{attribute 'linkalways'} 
{attribute 'no_explicit_call' := 'This FB is a CLASS and must be accessed using methods or properties'}
{attribute 'enable_dynamic_creation'}
FUNCTION_BLOCK Node_F_VN_ScharrFilter EXTENDS VisionNode
VAR
	ipSrcImage : _ITcVnImage;
    ipDestImage : _ITcVnImage;
    eDestDepth : _ETcVnElementType(ETcVnElementType.TCVN_ET_SAME_AS_SOURCE);
    eFilterDirection : _ETcVnFilterDirection(ETcVnFilterDirection.TCVN_FD_X);
    hrPrev : _HRESULT(S_OK);
	hresult : _HRESULT(S_OK);
END_VAR

METHOD PUBLIC  Clone : I_Node
VAR
	pNode : POINTER TO Node_F_VN_ScharrFilter;
END_VAR
pNode := __NEW(Node_F_VN_ScharrFilter);
Clone := pNode^;
END_METHOD

METHOD FB_init : BOOL
VAR_INPUT
	bInitRetains : BOOL; // if TRUE, the retain variables are initialized (warm start / cold start)
	bInCopyCode : BOOL;  // if TRUE, the instance afterwards gets moved into the copy code (online change)
END_VAR
AddInput('ipSrcImage', ipSrcImage);
AddParameter('eDestDepth', eDestDepth);
AddParameter('eFilterDirection', eFilterDirection);
AddInput('hrPrev', hrPrev);
AddOutput('ipDestImage', ipDestImage);
AddOutput('hresult',hresult);
END_METHOD

METHOD PROTECTED OnExecute
hresult.Value := F_VN_ScharrFilter(
	ipSrcImage:= ipSrcImage.Value,
	ipDestImage:= ipDestImage.Value,
	eDestDepth:= eDestDepth.Value,
	eFilterDirection:= eFilterDirection.Value,
	hrPrev:= hrPrev.Value);
END_METHOD

METHOD PUBLIC PreExecutionCheck
VAR_INPUT
	Check : I_PreExecutionChecks;
END_VAR
Check.IsTrue(ipSrcImage.IsValid, 'ipSrcImage must contain an image');
END_METHOD

END_FUNCTION_BLOCK

(* stored: Version 1.1.0.1, ProductVersion 3.1.4024.13
   POU Node_F_VN_ScharrFilter: Id {ad0601d1-7eab-0422-2102-390014244837}, SpecialFunc None
   Folder Constructor: Id {a2aec7ab-c3ca-0a43-17fc-fb6aabda11f7}
   Method Clone: Id {82440fd2-9144-0066-1600-f8af81e030e4}
   Method FB_init: Id {dc7e1af3-22ee-0482-29bf-0f0f7b019185}
   Method OnExecute: Id {3da6fe4c-7258-0c38-1e7c-ea8323a36f2b}
   Method PreExecutionCheck: Id {db6fc90c-b05a-0cee-3073-2784a9d4040a} *)
